PROGRAM Sample_ModbusRTU
VAR
	ModbusRTU				: FB_ModbusRTU;
	MesBlock				: ARRAY[1..8] OF ARRAY[1..120] OF WORD;	
	AX_Addr					: ARRAY[1..8] OF UINT 	:= [1,		1,		1,		1,		1, 		1, 		1, 		1];
	AX_Qty					: ARRAY[1..8] OF UINT	:= [1,		1,		1,		1,		1, 		1, 		1, 		1];
	AX_UnitId				: ARRAY[1..8] OF BYTE	:= [1,		1,		1,		1,		1, 		1, 		1, 		1];
	AX_Function				: ARRAY[1..8] OF UINT	:= [1,		2,		3,		4,		5, 	 	6, 	 	15, 	16];	
	AX_Priority				: ARRAY[1..8] OF UINT	:= [1,		1,		1,		1,		1, 	 	1, 	 	1, 		1 ];
	AX_bStart				: ARRAY[1..8] OF BOOL;
	MbStruct				: ARRAY[1..8] OF Struct_InputRTU;	
	
	KK: INT;
END_VAR

ModbusRTU();

FOR KK := 1 TO 8 DO 
	MbStruct[KK].InBuffer := ADR(MesBlock[KK]);
	MbStruct[KK].InFunction := AX_Function[KK];
	MbStruct[KK].InQuantity := AX_Qty[KK];
	MbStruct[KK].InStartAddr := AX_Addr[KK];
	MbStruct[KK].InUnitID := AX_UnitId[KK];
END_FOR


IF CalLocalTimeStruct.wSecond MOD 5 = 0 THEN
	FOR KK := 1 TO 8 DO
		IF AX_bStart[KK] THEN
			ModbusRTU.M_AddAction_FIFO(InStruct := MbStruct[KK], InPriority := AX_Priority[KK]);
		END_IF
	END_FOR
	
END_IF

END_PROGRAM

(* stored: Version 1.1.0.1, ProductVersion 3.1.4024.6
   POU Sample_ModbusRTU: Id {fa908d49-0b00-4312-9c25-9f23e27c9b20}, SpecialFunc None *)
